// TIA Portal V20 export
TYPE "LER_typeCommunicationReelCut"
// stored: Access Published
   STRUCT
      ReelCutToStack : "LER_typeCommunicationDataR2S";
      StackToReelCut : "LER_typeCommunicationDataS2R";
   END_STRUCT;
END_TYPE
